VAR_GLOBAL CONSTANT
    OPENED         	: DWORD := 16#0001;
    CLOSED         	: DWORD := 16#0002;
    SHORT_CIRCUIT   : DWORD := 16#0010;
    OPEN_CIRCUIT    : DWORD := 16#0020;
    STATUS_FAULT_OVERRIDE : DWORD := 16#0040;
END_VAR

(* stored: Version 1.1.0.1, ProductVersion 3.1.4024.15
   GVL GVL_ValveStatus: Id {59ad9f5b-4d90-436d-b338-fc83937e29c2} *)
